# B&R Automation Studio project HelloIO
Automation Studio 4.9

## Configuration Config1

CPU X20CP1686X, AutomationRuntime 6.2.1, Build 11.3.0, Vc 6.0.0

### Task classes (Cpu.sw)
```
Cyclic#4:
  HelloIO <- HelloIO.prg
```

### Hardware
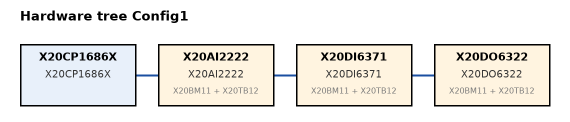
```
X20AI2222 : X20AI2222 v1.4.0.0  [SS1 -> X20TB12.SS; SL -> X20BM11.SL1]
X20BM11 : X20BM11 v1.1.0.0  [X2X1 -> X20CP1686X.IF6]
X20BM11_a : X20BM11 v1.1.0.0  [X2X1 -> X20BM11.X2X2]
X20BM11_b : X20BM11 v1.1.0.0  [X2X1 -> X20BM11_a.X2X2]
X20CP1686X : X20CP1686X v1.8.2.0
  Connector IF2:
    ActivateDevice = 1
    Mode = Manual
    InternetAddress = 192.168.1.50
    SubnetMask = 255.255.255.0
    ActivateSnmp = 2
  ConfigurationID = HelloIO_Config1
  FileDevice1
  FileDeviceName1 = USER
  FileDevicePath1 = USER_PATH
X20DI6371 : X20DI6371 v1.2.2.0  [SS1 -> X20TB12_a.SS; SL -> X20BM11_a.SL1]
X20DO6322 : X20DO6322 v1.4.1.0  [SS1 -> X20TB12_b.SS; SL -> X20BM11_b.SL1]
X20TB12 : X20TB12 v1.0.0.0
X20TB12_a : X20TB12 v1.0.0.0
X20TB12_b : X20TB12 v1.0.0.0
```

### IoMap.iom - X20CP1686X/IoMap.iom
```iecst
VAR_CONFIG
	::HelloIO:do1 AT %QX."X20DO6322".DigitalOutput01;
	::HelloIO:do2 AT %QX."X20DO6322".DigitalOutput02;
	::HelloIO:do3 AT %QX."X20DO6322".DigitalOutput03;
	::HelloIO:do4 AT %QX."X20DO6322".DigitalOutput04;
	::HelloIO:do5 AT %QX."X20DO6322".DigitalOutput05;
	::HelloIO:do6 AT %QX."X20DO6322".DigitalOutput06;
END_VAR
```

## Logical view

### Program Logical/HelloIO (IEC)

#### Variables.var
```iecst
VAR
	do1 : BOOL;
	do2 : BOOL;
	do3 : BOOL;
	do4 : BOOL;
	do5 : BOOL;
	do6 : BOOL;
	state : INT;
END_VAR
```

#### Main.st
```iecst
PROGRAM _INIT
	(* Insert code here *)

END_PROGRAM

PROGRAM _CYCLIC
	(* Insert code here *)
	do1 := FALSE;
	do2 := FALSE;
	do3 := FALSE;
	do4 := FALSE;
	do5 := FALSE;
	do6 := FALSE;

	CASE state OF
		0:
			do1 := TRUE;
			state := 5;
		5:
			do2 := TRUE;
			state := 10;
		10:
			do3 := TRUE;
			state := 15;
		15:
			do4 := TRUE;
			state := 20;
		20:
			do5 := TRUE;
			state := 25;
		25:
			do6 := TRUE;
			state := 0;
	END_CASE

END_PROGRAM

PROGRAM _EXIT
	(* Insert code here *)

END_PROGRAM
```

Listed in the project but not available here: Logical/Global.typ, Logical/Global.var, Logical/Libraries
